{attribute 'qualified_only'}
{attribute 'strict'}
{attribute 'to_string'}
TYPE E_CraneStatus :
(
	Off := 0,
	On := 1,
	Ready := 2,
	Running := 3
);
END_TYPE

(* stored: Version 1.1.0.1, ProductVersion 3.1.4026.12
   DUT E_CraneStatus: Id {310e15ef-4538-432e-a625-f05c35eaa75f} *)
